FUNCTION F_HigherValue : REAL
VAR_INPUT
	Value1																: REAL;
	Value2																: REAL;
END_VAR
VAR
END_VAR

// F_HigherValue
// Rev 1.0 - February 25, 2024

F_HigherValue															:= SEL(Value1 > Value2, Value2, Value1);

END_FUNCTION

(* stored: Version 1.1.0.1, ProductVersion 3.1.4024.12
   POU F_HigherValue: Id {1be1d932-f41b-4781-9a77-262a21528b4e}, SpecialFunc None *)
